FUNCTION_BLOCK FB_Positionsregler
VAR_INPUT
	targetPos		: sPosition;
	actualPos		: sPosition;
END_VAR
VAR_OUTPUT
	vXCartesianToMotors		: LREAL :=0;
	vYCartesianToMotors		: LREAL :=0;
	vThetaCartesianToMotors	: LREAL :=0;
END_VAR
VAR
	error		: sPosition;	// Positionsfehler
	deltaError	: sPosition;	// Fehlersteigung

	// Geschwindigkeit in Weltkoordinaten 
	W_X_targetSpeed		: LREAL; 
	W_Y_targetSpeed		: LREAL; 
	W_Theta_targetSpeed : LREAL;
	
	// Geschwindigkeit in Roboterkoordinaten
	R_X_targetSpeed		: LREAL;
	R_Y_targetSpeed		: LREAL;
	R_Theta_targetSpeed	: LREAL;
	
	// Reglerparameter
	KPX		: LREAL 	:= 0.2;
	KPY		: LREAL		:= 0.2;
	KPTheta	: LREAL 	:= 0.3;
	
	speedThreshold	: LREAL := 0.01; //Annäherung nur aktiv bei Abweichung > threshold
	AccelerationRate: LREAL := 5; 	//Höhere Werte = höhere Beschleunigung
	
	// Fuzzy Calkulation
	MembershipE : ARRAY[1..5] OF LREAL;
	MembershipDE : ARRAY[1..5] OF LREAL;
	i: INT;
	j: INT;
	ruleIdx: INT;
	weight: LREAL;
	numerator : LREAL := 0.0;
	denominator : LREAL := 0.0;
	initDone: BOOL := FALSE;
	
	RuleTable : ARRAY[1..5, 1..5] OF INT;
	OutputValue : ARRAY[1..5] OF REAL := [
        0.0,   // ZS
        0.25,  // PS
        0.5,   // PM
        0.75,  // PL
        1.0    // HL
    ];
	oldErrorTheta: LREAL;
END_VAR

// Wollte ich eigentlich oben machen, aber wollte er iwie nicht. Auf dauer noch ändern
IF NOT initDone THEN
    // RuleTable initialisieren (Zeile-für-Zeile), vermeidet statische Literal-Initialisierung
    RuleTable[1,1] := 5; RuleTable[1,2] := 5; RuleTable[1,3] := 4; RuleTable[1,4] := 4; RuleTable[1,5] := 3;
    RuleTable[2,1] := 4; RuleTable[2,2] := 4; RuleTable[2,3] := 4; RuleTable[2,4] := 3; RuleTable[2,5] := 2;
    RuleTable[3,1] := 4; RuleTable[3,2] := 4; RuleTable[3,3] := 3; RuleTable[3,4] := 2; RuleTable[3,5] := 4;
    RuleTable[4,1] := 4; RuleTable[4,2] := 3; RuleTable[4,3] := 2; RuleTable[4,4] := 2; RuleTable[4,5] := 1;
    RuleTable[5,1] := 3; RuleTable[5,2] := 2; RuleTable[5,3] := 2; RuleTable[5,4] := 1; RuleTable[5,5] := 1;

    OutputValue[1] := 0.0;
    OutputValue[2] := 0.25;
    OutputValue[3] := 0.5;
    OutputValue[4] := 0.75;
    OutputValue[5] := 1.0;
    initDone := TRUE;
END_IF

// --------------------------------------------------
// Winkelfehlerberechnung (Theta)
// --------------------------------------------------

// Winkelabweichung zwischen Soll und Ist berechnen
error.reWinkel := targetPos.reWinkel - actualPos.reWinkel;

// Normierung der Winkelabweichung auf den Bereich [-PI, PI]
// → stellt sicher, dass immer der kürzeste Drehweg verwendet wird
IF error.reWinkel > PI THEN
    error.reWinkel := error.reWinkel - 2.0 * PI;
ELSIF error.reWinkel < -PI THEN
    error.reWinkel := error.reWinkel + 2.0 * PI;
END_IF;

// Alten Fehlerwert für die Ableitung speichern
oldErrorTheta := error.reWinkel;

// Aktuellen Winkelfehler setzen
// Vorzeichen ggf. an Drehrichtungskonvention anpassen
error.reWinkel := -error.reWinkel;

// Änderung des Fehlers (D-Anteil)
deltaError.reWinkel := error.reWinkel - oldErrorTheta;


// --------------------------------------------------
// Positionsfehlerberechnung (X, Y)
// --------------------------------------------------

// Fehleränderung berechnen (Differenz zum vorherigen Fehler)
deltaError.reX := error.reX - (targetPos.reX - actualPos.reX);
deltaError.reY := error.reY - (targetPos.reY - actualPos.reY);

// Aktuellen Positionsfehler berechnen
error.reX := targetPos.reX - actualPos.reX;
error.reY := targetPos.reY - actualPos.reY;

// --------------------------------------------------
// Positionsregelung
// --------------------------------------------------

// ACT_GetFuzzyParam();

// Berechnung der Stellgröße
W_X_targetSpeed 	:= (error.reX 		* KPX);
W_Y_targetSpeed 	:= (error.reY 		* KPY);
W_Theta_targetSpeed := (error.reWinkel 	* KPTheta);

// Umrechnung von Welt in Motorcoordinaten
R_X_targetSpeed 	:= W_X_targetSpeed * COS(actualPos.reWinkel) - W_Y_targetSpeed * SIN(actualPos.reWinkel);
R_Y_targetSpeed 	:= W_Y_targetSpeed * COS(actualPos.reWinkel) + W_X_targetSpeed * SIN(actualPos.reWinkel);
R_Theta_targetSpeed := W_Theta_targetSpeed;

ACT_LimitACC();

ACTION ACT_GetFuzzyParam:
// Berechnen des Kx Reglers
METH_InputMembership(e := error.reX, outArr := MembershipE);
METH_InputMembership(e := deltaError.reX, outArr := MembershipDE);

// Defuzzyfication
FOR i := 1 TO 5 DO
    FOR j := 1 TO 5 DO
        weight := MembershipE[i] * MembershipDE[j];
        ruleIdx := RuleTable[i,j];

        numerator := numerator + weight * OutputValue[ruleIdx];
        denominator := denominator + weight;
    END_FOR
END_FOR

IF denominator > 0 THEN
    KPX := numerator / denominator;
ELSE
    KPX := 0.0; // fallback
END_IF

// Berechnen des Ky Reglers
METH_InputMembership(e := error.reY, 		outArr := MembershipE);
METH_InputMembership(e := deltaError.reY, 	outArr := MembershipDE);

// Defuzzyfication
FOR i := 1 TO 5 DO
    FOR j := 1 TO 5 DO
        weight := MembershipE[i] * MembershipDE[j];
        ruleIdx := RuleTable[i,j];

        numerator := numerator + weight * OutputValue[ruleIdx];
        denominator := denominator + weight;
    END_FOR
END_FOR

IF denominator > 0 THEN
    KPY := numerator / denominator;
ELSE
    KPY := 0.0; // fallback
END_IF
END_ACTION

ACTION ACT_LimitACC:
//Smoothes Annähern an den Sollwert, anpassbar über integrationRate
// x Werte 
IF ABS(vXCartesianToMotors - R_X_targetSpeed) > speedThreshold THEN   
    IF vXCartesianToMotors < R_X_targetSpeed THEN
        vXCartesianToMotors := vXCartesianToMotors + AccelerationRate * 0.01;  //Beschleunigung vorwärts
    ELSE
        vXCartesianToMotors := vXCartesianToMotors - AccelerationRate * 0.01;  //Beschleunigung rückwärts
    END_IF
END_IF
// y Werte 
IF ABS(vYCartesianToMotors - R_Y_targetSpeed) > speedThreshold THEN   
    IF vYCartesianToMotors < R_Y_targetSpeed THEN
        vYCartesianToMotors := vYCartesianToMotors + AccelerationRate * 0.01;  //Beschleunigung vorwärts
    ELSE
        vYCartesianToMotors := vYCartesianToMotors - AccelerationRate * 0.01;  //Beschleunigung rückwärts
    END_IF
END_IF
// Theta Werte 
IF ABS(vThetaCartesianToMotors - R_Theta_targetSpeed) > speedThreshold THEN   
    IF vThetaCartesianToMotors < R_Theta_targetSpeed THEN
        vThetaCartesianToMotors := vThetaCartesianToMotors + AccelerationRate * 0.01;  //Beschleunigung vorwärts
    ELSE
       vThetaCartesianToMotors := vThetaCartesianToMotors - AccelerationRate * 0.01;  //Beschleunigung rückwärts
    END_IF
END_IF
END_ACTION

METHOD METH_InputMembership
VAR_INPUT
	e	: LREAL;
END_VAR
VAR_IN_OUT
	outArr : ARRAY[1..5] OF LREAL;
END_VAR
// einfache dreieckige Memberships als Beispiel (anpassen an deine MF)
outArr[1] := MAX(0.0, ( -e - 0.5) / 0.5);      // NL (links)
outArr[2] := MAX(0.0, 1.0 - ABS(e + 0.5) / 0.75); // NS
outArr[3] := MAX(0.0, 1.0 - ABS(e) / 1.0);       // ZE
outArr[4] := MAX(0.0, 1.0 - ABS(e - 0.5) / 0.75); // PS
outArr[5] := MAX(0.0, (e - 0.5) / 0.5);        // PL
END_METHOD

END_FUNCTION_BLOCK

(* stored: Version 1.1.0.1, ProductVersion 3.1.4026.13
   POU FB_Positionsregler: Id {5eaf5f69-503a-4e20-898f-d897551e6b9b}, SpecialFunc None
   Action ACT_GetFuzzyParam: Id {4ee22feb-6be5-4906-80b6-3d87f4f37582}
   Action ACT_LimitACC: Id {e1d0b9f1-bfb7-427c-a749-b6c6114fd6e7}
   Method METH_InputMembership: Id {8b1199f8-59f0-4cc6-be94-a8ade66a0e7f} *)
